// Mitsubishi GX Works2 project: WheelValveTapFX3S   PLC: FX3S

// global labels: Global1
VAR_GLOBAL
  XXLimitN AT M8344 : BOOL;
  XXLimitP AT M8343 : BOOL;
  XXBusy AT M8340 : BOOL;
  XXInterruptInverse AT M8347 : BOOL;
  XXPos AT D8340 : DINT;
  XXAccelTime AT D8348 : INT;
  XXDecelTime AT D8349 : INT;
  XXPosView AT D0 : DINT;
  XXTarPos AT D2 : DINT;
  XXFeed AT D4 : DINT;
  XXTarR AT M0 : BOOL;
  XXTarRSkip AT D6 : INT;
  XXOn AT M1 : BOOL;
  XXRun AT M2 : BOOL;
  XXDirection AT M3 : BOOL;
  XXMinI AT X000 : BOOL;
  XXMaxI AT X001 : BOOL;
  XXPulseO AT Y000 : BOOL;
  XXDirectionO AT Y004 : BOOL;
  XXOnO AT Y002 : BOOL;
  YYLimitN AT M8354 : BOOL;
  YYLimitP AT M8353 : BOOL;
  YYBusy AT M8350 : BOOL;
  YYInterruptInverse AT M8357 : BOOL;
  YYPos AT D8350 : DINT;
  YYAccelTime AT D8358 : INT;
  YYDecelTime AT D8359 : INT;
  YYPosView AT D7 : DINT;
  YYTarPos AT D9 : DINT;
  YYFeed AT D11 : DINT;
  YYTarR AT M4 : BOOL;
  YYTarRSkip AT D13 : INT;
  YYOn AT M5 : BOOL;
  YYRun AT M6 : BOOL;
  YYDirection AT M7 : BOOL;
  YYPulseO AT Y001 : BOOL;
  YYDirectionO AT Y005 : BOOL;
  YYOnO AT Y003 : BOOL;
  Run AT M8 : BOOL;
  RunStop AT M9 : BOOL;
  RunState AT D14 : INT;
  RunStateNext AT M10 : BOOL;
  RunSwitchI AT X002 : BOOL;
  Tap AT M11 : BOOL;
  TapI AT X003 : BOOL;
END_VAR

// task Task_01 (event TRUE, interval 0, priority 31): POU_01

PROGRAM POU_01
VAR
  fTmp : BOOL;
END_VAR
RST(M8002, XXOnO);
SET(M8002, YYOnO);
MOV(M8002, 200, XXAccelTime);
MOV(M8002, 200, XXDecelTime);
MOV(M8002, 200, YYAccelTime);
MOV(M8002, 200, YYDecelTime);
(*1000 pulse = 1 mm, 1000 pulse = 1 round, XX pulse = 0.79375 * YY pulse)
(*feed 40000 pps = 2400 rpm*)
(*|||||||||||||||*)
(*|||||||||||||||*)
SET(Run AND RunState = 0, fTmp);
MOV(fTmp, 1, RunState);
RST(fTmp, Run);
RST(fTmp, fTmp);
SET(RunStop, fTmp);
RST(fTmp, RunStop);
RST(fTmp, RunState);
RST(fTmp, XXRun);
RST(fTmp, YYRun);
RST(fTmp, fTmp);
(*|||||||||||||||*)
(*|||||||||||||||*)
INC(RunStateNext, RunState);
RST(M8000, RunStateNext);
DECO(M8000, RunState, 6, M100); DECO(M8000, RunState, 6, M1100); ZRST(NOT XXTarR OR NOT YYTarR, M1100, M1163);
(*|||||||||||||||*)
(*|||||||||||||||*)
(*/////get origin*)
(*at min, jump to move down*)
SET(M1101 AND XXMinI, fTmp);
MOV(fTmp, 3, RunState); RST(fTmp, fTmp);
(*not at min, move up*)
SET(M1101 AND NOT XXMinI, fTmp);
RST(fTmp, XXPos);
RST(fTmp, YYPos);
DMOV(fTmp, -45_000, XXTarPos);
DMOV(fTmp, -56_693, YYTarPos);
DMOV(fTmp, 10_000, XXFeed);
DMOV(fTmp, 12_598, YYFeed);
SET(fTmp, XXRun);
SET(fTmp, YYRun);
SET(fTmp, RunStateNext); RST(fTmp, fTmp);
(*move up hit limit, reset*)
SET(M102 AND NOT XXBusy AND NOT YYBusy, fTmp);
RST(fTmp, XXRun);
RST(fTmp, YYRun);
RST(fTmp, XXPos);
RST(fTmp, YYPos);
SET(fTmp, RunStateNext); RST(fTmp, fTmp);
(*move down*)
SET(M1103, fTmp);
DMOV(fTmp, 20_000, XXTarPos);
DMOV(fTmp, 1_000, XXFeed);
SET(fTmp, XXRun);
SET(fTmp, RunStateNext); RST(fTmp, fTmp);
(*move down out min, stop*)
SET(M104 AND NOT XXMinI, fTmp);
RST(fTmp, XXRun);
SET(fTmp, RunStateNext); RST(fTmp, fTmp);
(*stop done, move down 5mm*)
SET(M1105, fTmp);
DMOV(fTmp, XXPos + 5000, XXTarPos);
SET(fTmp, XXRun);
SET(fTmp, RunStateNext); RST(fTmp, fTmp);
(*move down 5mm done, ready*)
SET(M1106, fTmp);
RST(fTmp, XXPos);
RST(fTmp, YYPos);
MOV(fTmp, 11, RunState); RST(fTmp, fTmp);
(*/////main sequence*)
(*wait tap hit, move down fast*)
SET(M1111 AND Tap, fTmp);
RST(fTmp, Tap);
DMOV(fTmp, 15_000, XXTarPos);
DMOV(fTmp, 18_898, YYPos);
DMOV(fTmp, 50000, XXFeed);
SET(fTmp, XXRun);
SET(fTmp, RunStateNext); RST(fTmp, fTmp);
(*move down fast done, move down slow*)
SET(M1112, fTmp);
DMOV(fTmp, 45_000, XXTarPos);
DMOV(fTmp, 56_693, YYTarPos);
DMOV(fTmp, 25400, XXFeed);
DMOV(fTmp, 32000, YYFeed);
SET(fTmp, XXRun);
SET(fTmp, YYRun);
SET(fTmp, RunStateNext); RST(fTmp, fTmp);
(*move down slow done, move up*)
SET(M1113, fTmp);
DMOV(fTmp, 0, XXTarPos);
DMOV(fTmp, 0, YYTarPos);
DMOV(fTmp, 31750, XXFeed);
DMOV(fTmp, 40000, YYFeed);
SET(fTmp, XXRun);
SET(fTmp, YYRun);
SET(fTmp, RunStateNext); RST(fTmp, fTmp);
(*move up done, return wait tap hit*)
SET(M1114, fTmp);
MOV(fTmp, 11, RunState); RST(fTmp, fTmp);
(*|||||||||||||||*)
(*|||||||||||||||*)
(*XX*)
RST(XXRun AND XXTarPos = XXPos, XXRun);
DDRVA(XXRun, XXTarPos, XXFeed, XXPulseO, XXDirection);
RST(M8029, XXRun);
OUT(XXDirection, XXDirectionO);
INC(NOT XXRun AND NOT XXBusy AND XXTarRSkip < 5, XXTarRSkip);
RST(XXRun, XXTarRSkip);
OUT(XXTarRSkip >= 5, XXTarR);
(**)
OUT(XXMinI, XXLimitN);
OUT(XXMaxI, XXLimitP);
(*YY*)
RST(YYRun AND YYTarPos = YYPos, YYRun);
DDRVA(YYRun, YYTarPos, YYFeed, YYPulseO, YYDirection);
RST(M8029, YYRun);
OUT(YYDirection, YYDirectionO);
INC(NOT YYRun AND NOT YYBusy AND YYTarRSkip < 5, YYTarRSkip);
RST(YYRun, YYTarRSkip);
OUT(YYTarRSkip >= 5, YYTarR);
(**)
OUT(XXMinI, YYLimitN);
OUT(XXMaxI, YYLimitP);
(*|||||||||||||||*)
(*|||||||||||||||*)
PLS(RunSwitchI, Run); SET(Run, Run);
PLF(RunSwitchI, RunStop); SET(RunStop, RunStop);
PLS(TapI, Tap); SET(Tap, Tap);
(*|||||||||||||||*)
(*|||||||||||||||*)
END_PROGRAM
